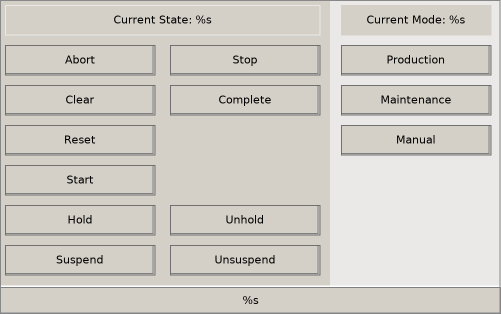
VISUALIZATION V_PackMLModule  // 501x314
VAR_IN_OUT
	PackML_HMI : ST_PackMLStatemachine_HMI;
END_VAR
    Rectangle (0,0 330x285)
    Textfield (5,5 315x30), "Current State: %s", text variable: PackML_HMI.CurrentState
    Button (5,45 150x30), "Abort"
        OnMouseClick: execute { PackML_HMI.StateCommand := E_PMLCommand.Abort; }
    Button (5,85 150x30), "Clear"
        OnMouseClick: execute { PackML_HMI.StateCommand := E_PMLCommand.Clear; }
    Button (5,125 150x30), "Reset"
        OnMouseClick: execute { PackML_HMI.StateCommand := E_PMLCommand.Reset; }
    Button (5,165 150x30), "Start"
        OnMouseClick: execute { PackML_HMI.StateCommand := E_PMLCommand.Start; }
    Button (170,85 150x30), "Complete"
        OnMouseClick: execute { PackML_HMI.StateCommand := E_PMLCommand.Complete; }
    Button (170,45 150x30), "Stop"
        OnMouseClick: execute { PackML_HMI.StateCommand := E_PMLCommand.Stop; }
    Button (5,205 150x30), "Hold"
        OnMouseClick: execute { PackML_HMI.StateCommand := E_PMLCommand.Hold; }
    Button (170,205 150x30), "Unhold"
        OnMouseClick: execute { PackML_HMI.StateCommand := E_PMLCommand.Unhold; }
    Button (5,245 150x30), "Suspend"
        OnMouseClick: execute { PackML_HMI.StateCommand := E_PMLCommand.Suspend; }
    Button (170,245 150x30), "Unsuspend"
        OnMouseClick: execute { PackML_HMI.StateCommand := E_PMLCommand.Unsuspend; }
    Rectangle (330,0 171x285)
    Textfield (341,5 150x30), "Current Mode: %s", text variable: PackML_HMI.CurrentMode
    Button (341,45 150x30), "Production"
        OnMouseClick: execute { PackML_HMI.ModeCommand := 1; }
    Button (341,85 150x30), "Maintenance"
        OnMouseClick: execute { PackML_HMI.ModeCommand := 2; }
    Button (341,125 150x30), "Manual"
        OnMouseClick: execute { PackML_HMI.ModeCommand := 3; }
    Textfield (0,287 501x27), "%s", text variable: PackML_HMI.Name
END_VISUALIZATION

(* stored: Version 1.1.0.1, ProductVersion 3.1.4026.18
   Visu V_PackMLModule: Id {c32c8a65-fc58-4ac9-add0-1a43b05ef57f} *)
